TYPE ST_HMI_Machine_Command :
STRUCT
	Start: BOOL;
	Stop: BOOL;
	Reset: BOOL;
	Abort: BOOL;
END_STRUCT
END_TYPE

(* stored: Version 1.1.0.1, ProductVersion 3.1.4024.12
   DUT ST_HMI_Machine_Command: Id {296a0ede-7e02-4456-a8c7-f6a39c971a41} *)
